{attribute addProperty BoxType "EL3612-0000-0016"}
{attribute addProperty Id "AI_Inputs_ChannelAT %I*ARRAY[0..8] OF AI_Inputs_Channel_513C0694176220WcStateAT %I*WcState_98A4DF7520.250InfoDataAT %I*InfoData_BC63D37F80100"}
{attribute addProperty CRC "4148475682"}
{attribute addProperty SizeInBites "258"}
{attribute addProperty SizeInBytes "32.25"}
TYPE EL3612_174E1636 :
STRUCT
	{attribute addProperty Name "AI_Inputs_Channel"}
	AI_Inputs_Channel : ARRAY[0..8] OF AI_Inputs_Channel_513C0694;
	{attribute addProperty Name "WcState"}
	WcState : WcState_98A4DF75;
	{attribute addProperty Name "InfoData"}
	InfoData : InfoData_BC63D37F;
END_STRUCT
END_TYPE

(* stored: Version 1.2.0.0, ProductVersion 3.1.4024.9
   DUT EL3612_174E1636: Id {a7f9c864-e098-4721-9df4-6d3a6186ae12} *)
